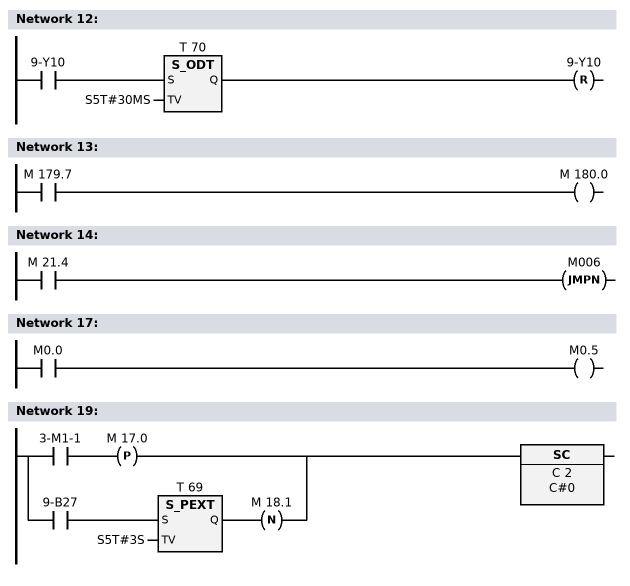
NETWORK
TITLE =
      A     "9-Y10";
      L     S5T#30MS;
      SD    T 70;
      NOP   0;
      NOP   0;
      NOP   0;
      A     T 70;
      R     "9-Y10";
NETWORK
TITLE =
      A     M 179.7;
      =     M 180.0;
NETWORK
TITLE =
      A     M 21.4;
      JCN   M006;
NETWORK
TITLE =
      L     MD 176;
      CAD;
      SLD   1;
      CAD;
      T     MD 176;
NETWORK
TITLE =
      L     MD 180;
      CAD;
      SLD   1;
      CAD;
      T     MD 180;
NETWORK
TITLE =
M006: A     "М0.0";
      =     "М0.5";
NETWORK
TITLE =
      A(;
      A     M 245.6;
      S     M 18.4;
      A(;
      O     "5-S11";
      O     M 245.3;
      ON    "М100.4";
      );
      R     M 18.4;
      A     M 18.4;
      );
      FN    M 18.2;
      R     M 18.0;
NETWORK
TITLE =
      A     "3-М1-1";
      FP    M 17.0;
      O(;
      A(;
      A     "9-В27";
      L     S5T#3S;
      SE    T 69;
      NOP   0;
      NOP   0;
      NOP   0;
      A     T 69;
      );
      FN    M 18.1;
      );
      L     C#0;
      S     C 2;
END_FUNCTION

FUNCTION FC 66 : VOID
AUTHOR : Stolz
VERSION : 0.1
BEGIN
// (block stored without names or comments; labels and parameter names are numbered)
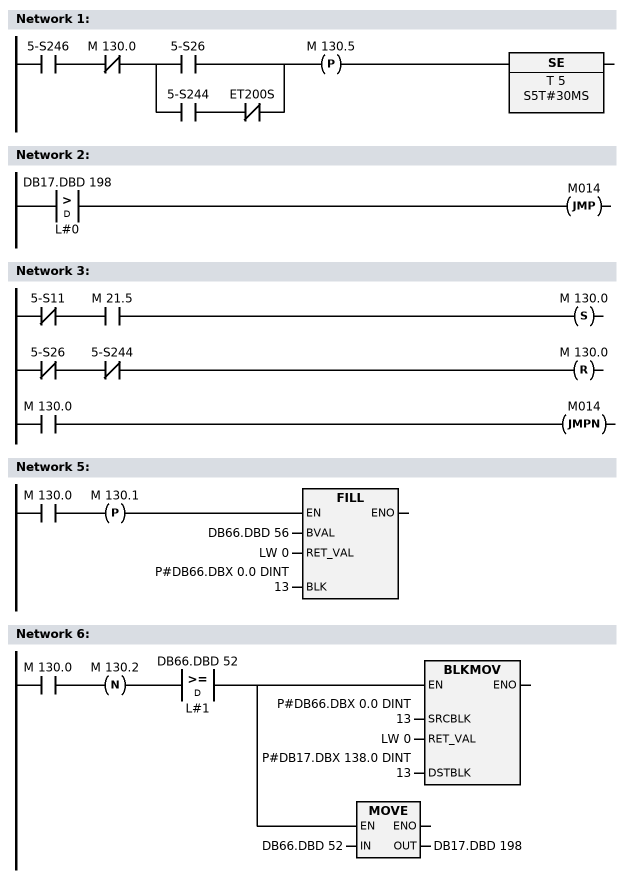
NETWORK
TITLE =
      A     "5-S246";
      AN    M 130.0;
      A(;
      O     "5-S26";
      O;
      A     "5-S244";
      AN    "ET200S";
      );
      FP    M 130.5;
      L     S5T#30MS;
      SE    T 5;
NETWORK
TITLE =
      L     DB17.DBD 198;
      L     L#0;
      >D;
      JC    M014;
NETWORK
TITLE =
      AN    "5-S11";
      A     M 21.5;
      S     M 130.0;
      AN    "5-S26";
      AN    "5-S244";
      R     M 130.0;
      A     M 130.0;
      JCN   M014;
NETWORK
TITLE =
      A     M 21.7;
      JCN   M001;
      L     C 10;
      ITD;
      T     DB66.DBD 0;
      L     L#0;
      T     DB66.DBD 52;
M001: A     M 22.0;
      JCN   M002;
      L     C 10;
      ITD;
      T     DB66.DBD 4;
      L     L#0;
      T     DB66.DBD 52;
M002: A     M 22.1;
      JCN   M003;
      L     C 10;
      ITD;
      T     DB66.DBD 8;
      L     L#0;
      T     DB66.DBD 52;
M003: A     M 22.2;
      JCN   M004;
      L     C 10;
      ITD;
      T     DB66.DBD 12;
      L     L#0;
      T     DB66.DBD 52;
M004: A     M 22.3;
      JCN   M005;
      L     C 10;
      ITD;
      T     DB66.DBD 16;
      L     L#0;
      T     DB66.DBD 52;
M005: A     M 22.4;
      JCN   M006;
      L     C 10;
      ITD;
      T     DB66.DBD 20;
      L     L#0;
      T     DB66.DBD 52;
M006: A     M 22.5;
      JCN   M007;
      L     C 10;
      ITD;
      T     DB66.DBD 24;
      L     L#0;
      T     DB66.DBD 52;
M007: A     M 24.0;
      JCN   M008;
      L     C 10;
      ITD;
      T     DB66.DBD 28;
      L     L#0;
      T     DB66.DBD 52;
M008: A     M 24.1;
      JCN   M009;
      L     C 10;
      ITD;
      T     DB66.DBD 32;
      L     L#0;
      T     DB66.DBD 52;
M009: A     M 24.2;
      JCN   M010;
      L     C 10;
      ITD;
      T     DB66.DBD 36;
      L     L#0;
      T     DB66.DBD 52;
M010: A     M 24.3;
      JCN   M011;
      L     C 10;
      ITD;
      T     DB66.DBD 40;
      L     L#0;
      T     DB66.DBD 52;
M011: A     M 24.4;
      JCN   M012;
      L     C 10;
      ITD;
      T     DB66.DBD 44;
      L     L#0;
      T     DB66.DBD 52;
M012: A     M 24.5;
      JCN   M013;
      L     C 10;
      ITD;
      T     DB66.DBD 48;
      L     L#0;
      T     DB66.DBD 52;
M013: A     M 21.6;
      JCN   M014;
      L     C 10;
      ITD;
      T     DB66.DBD 52;
NETWORK
TITLE =
M014: A     M 130.0;
      FP    M 130.1;
      JNB   M015;
      CALL  "FILL" (
           BVAL                     := DB66.DBD 56,
           RET_VAL                  := LW 0,
           BLK                      := P#DB66.DBX 0.0 DINT 13);
M015: NOP   0;
NETWORK
TITLE =
      A     M 130.0;
      FN    M 130.2;
      A(;
      L     DB66.DBD 52;
      L     L#1;
      >=D;
      );
      =     L 2.0;
      A     L 2.0;
      JNB   M016;
      CALL  "BLKMOV" (
           SRCBLK                   := P#DB66.DBX 0.0 DINT 13,
           RET_VAL                  := LW 0,
           DSTBLK                   := P#DB17.DBX 138.0 DINT 13);
M016: NOP   0;
      A     L 2.0;
      JNB   M017;
      L     DB66.DBD 52;
      T     DB17.DBD 198;
M017: NOP   0;
END_FUNCTION

FUNCTION FC 100 : VOID
AUTHOR : Stolz
VERSION : 0.1
BEGIN
// (block stored without names or comments; labels and parameter names are numbered)
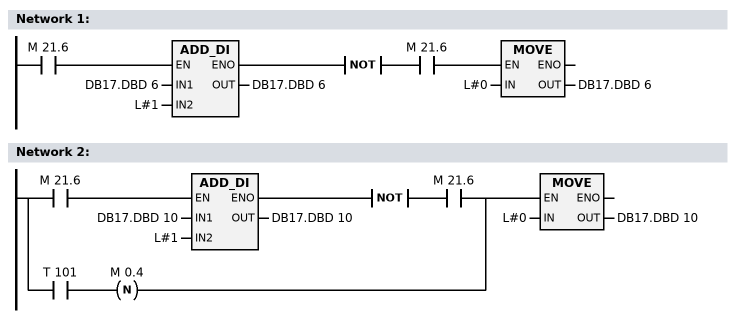
NETWORK
TITLE =
      A(;
      A     M 21.6;
      JNB   M001;
      L     DB17.DBD 6;
      L     L#1;
      +D;
      T     DB17.DBD 6;
      AN    OV;
      SAVE;
      CLR;
M001: A     BR;
      );
      NOT;
      A     M 21.6;
      JNB   M002;
      L     L#0;
      T     DB17.DBD 6;
M002: NOP   0;
NETWORK
TITLE =
      A(;
      A(;
      A     M 21.6;
      JNB   M003;
      L     DB17.DBD 10;
      L     L#1;
      +D;
      T     DB17.DBD 10;
      AN    OV;
      SAVE;
      CLR;
M003: A     BR;
      );
      NOT;
      A     M 21.6;
      O(;
      A     T 101;
      FN    M 0.4;
      );
      );
      JNB   M004;
      L     L#0;
      T     DB17.DBD 10;
M004: NOP   0;
END_FUNCTION

FUNCTION FC 104 : VOID
AUTHOR : Stolz
NAME : IstUmin
VERSION : 0.1
BEGIN
// (block stored without names or comments; labels and parameter names are numbered)
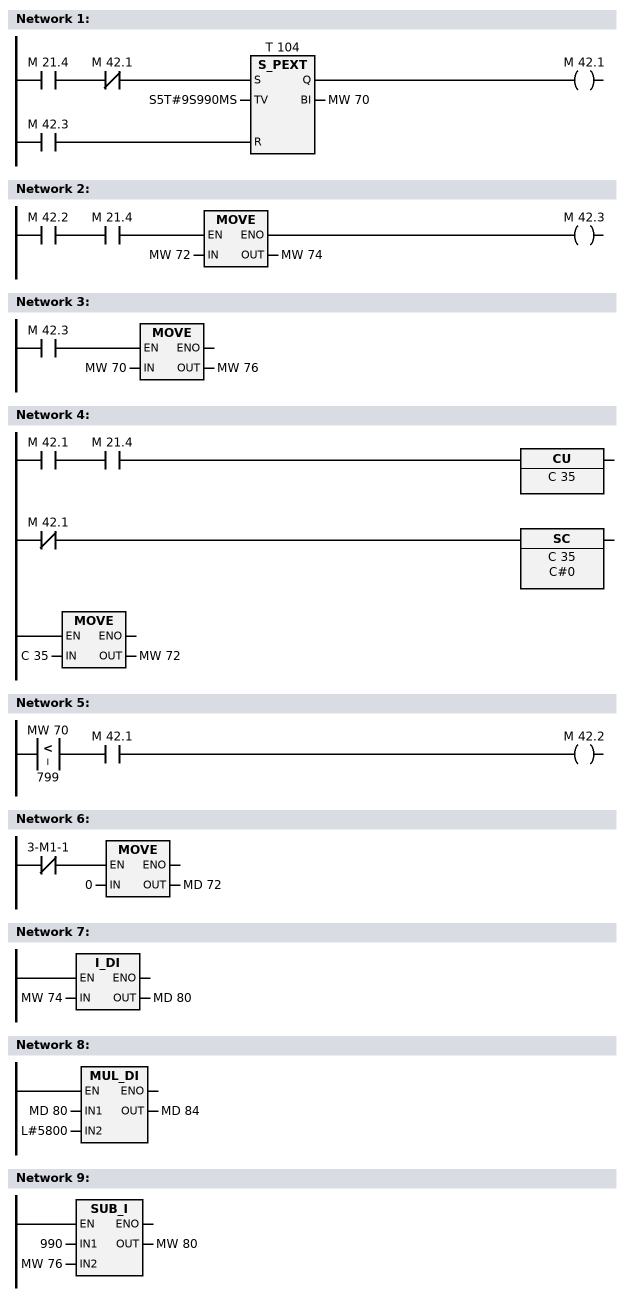
NETWORK
TITLE =
      A     M 21.4;
      AN    M 42.1;
      L     S5T#9S990MS;
      SE    T 104;
      A     M 42.3;
      R     T 104;
      L     T 104;
      T     MW 70;
      NOP   0;
      A     T 104;
      =     M 42.1;
NETWORK
TITLE =
      A     M 42.2;
      A     M 21.4;
      JNB   M001;
      L     MW 72;
      T     MW 74;
      SET;
      SAVE;
      CLR;
M001: A     BR;
      =     M 42.3;
NETWORK
TITLE =
      A     M 42.3;
      JNB   M002;
      L     MW 70;
      T     MW 76;
M002: NOP   0;
NETWORK
TITLE =
      A     M 42.1;
      A     M 21.4;
      CU    C 35;
      BLD   101;
      AN    M 42.1;
      L     C#0;
      S     C 35;
      NOP   0;
      L     C 35;
      T     MW 72;
      NOP   0;
      NOP   0;
NETWORK
TITLE =
      A(;
      L     MW 70;
      L     799;
      <I;
      );
      A     M 42.1;
      =     M 42.2;
NETWORK
TITLE =
      AN    "3-М1-1";
      JNB   M003;
      L     0;
      T     MD 72;
M003: NOP   0;
NETWORK
TITLE =
      L     MW 74;
      ITD;
      T     MD 80;
      NOP   0;
NETWORK
TITLE =
      L     MD 80;
      L     L#5800;
      *D;
      T     MD 84;
      NOP   0;
NETWORK
TITLE =
      L     990;
      L     MW 76;
      -I;
      T     MW 80;
      NOP   0;
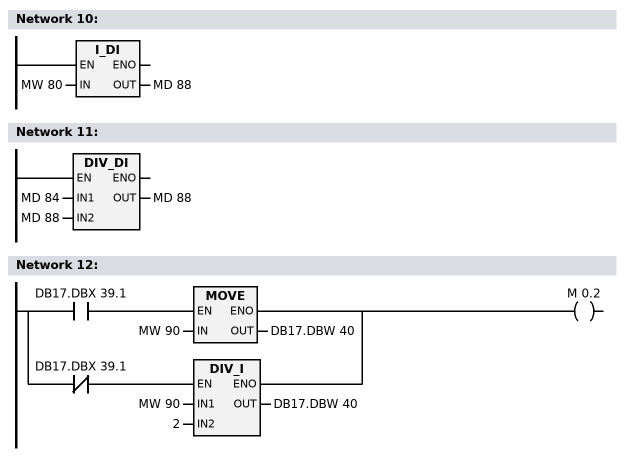
NETWORK
TITLE =
      L     MW 80;
      ITD;
      T     MD 88;
      NOP   0;
NETWORK
TITLE =
      L     MD 84;
      L     MD 88;
      /D;
      T     MD 88;
      NOP   0;
NETWORK
TITLE =
      O(;
      A     DB17.DBX 39.1;
      JNB   M004;
      L     MW 90;
      T     DB17.DBW 40;
      SET;
      SAVE;
      CLR;
M004: A     BR;
      );
      O(;
      AN    DB17.DBX 39.1;
      JNB   M005;
      L     MW 90;
      L     2;
      /I;
      T     DB17.DBW 40;
      AN    OV;
      SAVE;
      CLR;
M005: A     BR;
      );
      =     M 0.2;
END_FUNCTION

FUNCTION FC 105 : VOID
AUTHOR : Stolz
NAME : SollUmin
VERSION : 0.2
VAR_TEMP
  TEMP0 : INT ;
  TEMP1 : DINT ;
  TEMP2 : DINT ;
  TEMP3 : DINT ;
  TEMP4 : INT ;
  TEMP5 : DINT ;
  TEMP6 : DINT ;
  TEMP7 : DINT ;
END_VAR
BEGIN
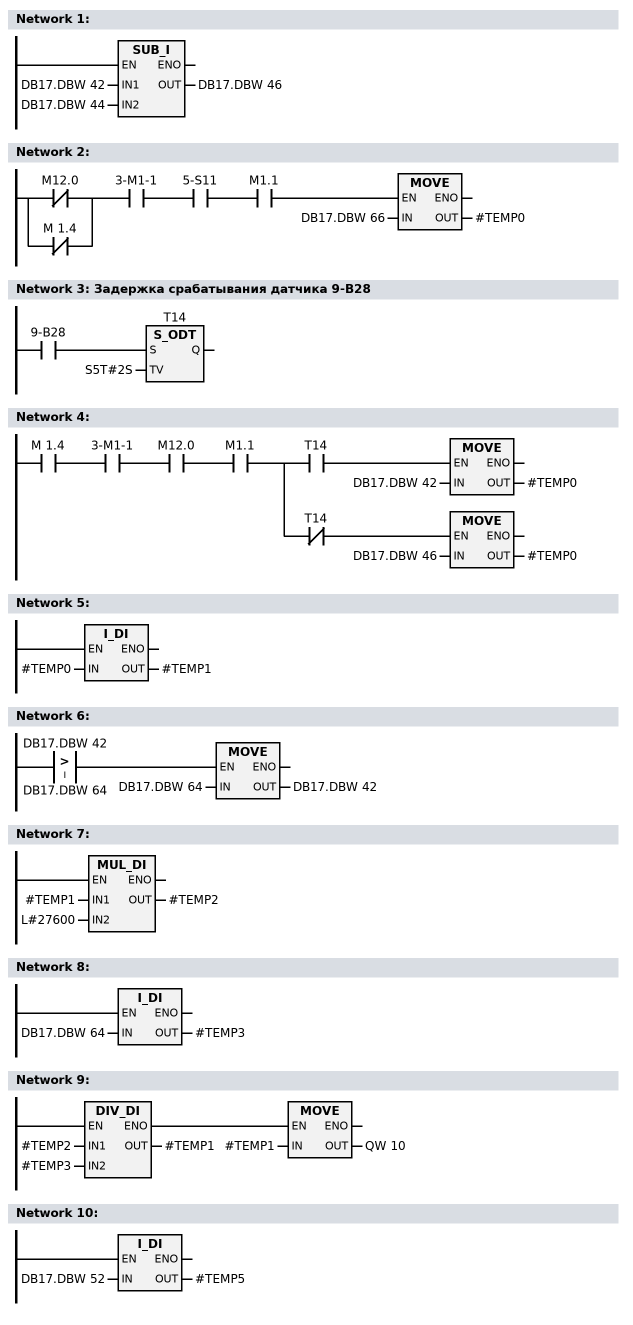
NETWORK
TITLE =
      L     DB17.DBW 42;
      L     DB17.DBW 44;
      -I;
      T     DB17.DBW 46;
      NOP   0;
NETWORK
TITLE =
      A(;
      ON    "М12.0";
      ON    M 1.4;
      );
      A     "3-М1-1";
      A     "5-S11";
      A     "М1.1";
      JNB   _001;
      L     DB17.DBW 66;
      T     #TEMP0;
_001: NOP   0;
NETWORK
TITLE = Задержка срабатывания датчика 9-В28
      A     "9-В28";
      L     S5T#2S;
      SD    "Т14";
      NOP   0;
      NOP   0;
      NOP   0;
      NOP   0;
NETWORK
TITLE =
      A     M 1.4;
      A     "3-М1-1";
      A     "М12.0";
      A     "М1.1";
      =     L 28.0;
      A     L 28.0;
      A     "Т14";
      JNB   _002;
      L     DB17.DBW 42;
      T     #TEMP0;
_002: NOP   0;
      A     L 28.0;
      AN    "Т14";
      JNB   _003;
      L     DB17.DBW 46;
      T     #TEMP0;
_003: NOP   0;
NETWORK
TITLE =
      L     #TEMP0;
      ITD;
      T     #TEMP1;
      NOP   0;
NETWORK
TITLE =
      A(;
      L     DB17.DBW 42;
      L     DB17.DBW 64;
      >I;
      );
      JNB   _004;
      L     DB17.DBW 64;
      T     DB17.DBW 42;
_004: NOP   0;
NETWORK
TITLE =
      L     #TEMP1;
      L     L#27600;
      *D;
      T     #TEMP2;
      NOP   0;
NETWORK
TITLE =
      L     DB17.DBW 64;
      ITD;
      T     #TEMP3;
      NOP   0;
NETWORK
TITLE =
      A(;
      L     #TEMP2;
      L     #TEMP3;
      /D;
      T     #TEMP1;
      AN    OV;
      SAVE;
      CLR;
      A     BR;
      );
      JNB   _005;
      L     #TEMP1;
      T     QW 10;
_005: NOP   0;
NETWORK
TITLE =
      L     DB17.DBW 52;
      ITD;
      T     #TEMP5;
      NOP   0;
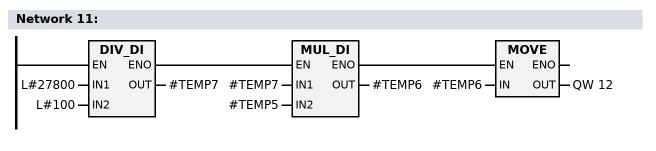
NETWORK
TITLE =
      A(;
      A(;
      L     L#27800;
      L     L#100;
      /D;
      T     #TEMP7;
      AN    OV;
      SAVE;
      CLR;
      A     BR;
      );
      JNB   _006;
      L     #TEMP7;
      L     #TEMP5;
      *D;
      T     #TEMP6;
      AN    OV;
      SAVE;
      CLR;
_006: A     BR;
      );
      JNB   _007;
      L     #TEMP6;
      T     QW 12;
_007: NOP   0;
END_FUNCTION

FUNCTION FC 110 : VOID
AUTHOR : Joehring
VERSION : 0.1
BEGIN
// (block stored without names or comments; labels and parameter names are numbered)
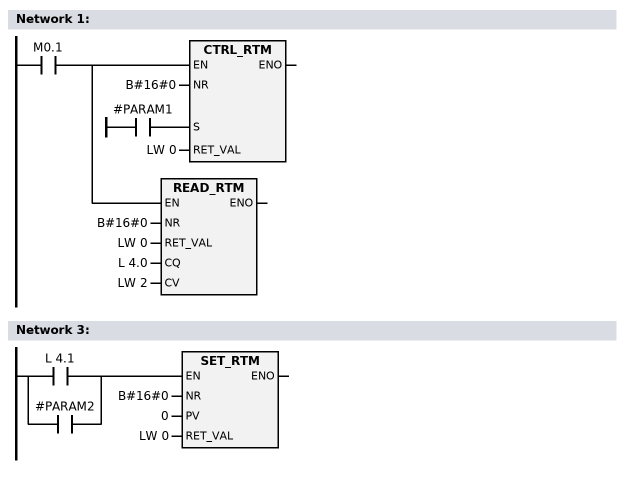
NETWORK
TITLE =
      A     "М0.1";
      =     L 5.0;
      A     #PARAM1;
      =     L 5.1;
      BLD   103;
      A     L 5.0;
      JNB   M001;
      CALL  "CTRL_RTM" (
           NR                       := B#16#0,
           S                        := L 5.1,
           RET_VAL                  := LW 0);
M001: NOP   0;
      A     L 5.0;
      JNB   M002;
      CALL  "READ_RTM" (
           NR                       := B#16#0,
           RET_VAL                  := LW 0,
           CQ                       := L 4.0,
           CV                       := LW 2);
M002: NOP   0;
NETWORK
TITLE =
      L     LW 2;
      L     1;
      >=I;
      =     L 4.1;
NETWORK
TITLE =
      A(;
      O     L 4.1;
      O     #PARAM2;
      );
      JNB   M003;
      CALL  "SET_RTM" (
           NR                       := B#16#0,
           PV                       := 0,
           RET_VAL                  := LW 0);
M003: NOP   0;
NETWORK
TITLE =
      O(;
      A     L 4.1;
      JNB   M004;
      L     #PARAM3;
      L     L#1;
      +D;
      T     #PARAM3;
      AN    OV;
      SAVE;
      CLR;
M004: A     BR;
      );
      O(;
      A     #PARAM2;
      JNB   M005;
      L     0;
      T     #PARAM3;
      SET;
      SAVE;
      CLR;
M005: A     BR;
      );
      =     L 4.2;
END_FUNCTION

// FC 125: know-how protected block, not included

DATA_BLOCK DB 17
AUTHOR : Stolz
VERSION : 0.2
BEGIN
// 360 bytes; values not shown
END_DATA_BLOCK

DATA_BLOCK DB 66
AUTHOR : Stolz
VERSION : 0.0
BEGIN
// 60 bytes; values not shown
END_DATA_BLOCK

DATA_BLOCK DB 77
AUTHOR : Stolz
VERSION : 0.0
BEGIN
// 80 bytes; values not shown
END_DATA_BLOCK

DATA_BLOCK DB 100
AUTHOR : Joehring
VERSION : 0.1
FB 100
BEGIN
END_DATA_BLOCK

DATA_BLOCK DB 111
VERSION : 0.1
BEGIN
// 88 bytes; values not shown
END_DATA_BLOCK

DATA_BLOCK DB 125
VERSION : 0.0
FB 125
BEGIN
END_DATA_BLOCK

ORGANIZATION_BLOCK OB 1
AUTHOR : Stolz
VERSION : 0.1
BEGIN
// (block stored without names or comments; labels and parameter names are numbered)
NETWORK
TITLE =
      UC    FC 50;
NETWORK
TITLE =
      UC    "FC2";
NETWORK
TITLE =
      UC    "FC3";
NETWORK
TITLE =
      UC    "FC4";
NETWORK
TITLE =
      UC    "FC6";
NETWORK
TITLE =
      UC    "FC7";
NETWORK
TITLE =
      UC    FC 10;
NETWORK
TITLE =
      UC    FC 11;
NETWORK
TITLE =
      UC    FC 12;
NETWORK
TITLE =
      UC    FC 23;
NETWORK
TITLE =
      UC    FC 24;
NETWORK
TITLE =
      UC    FC 60;
NETWORK
TITLE =
      A     DB17.DBX 39.3;
      CC    FC 61;
NETWORK
TITLE =
      UC    FC 100;
NETWORK
TITLE =
      UC    FC 104;
NETWORK
TITLE =
      UC    FC 105;
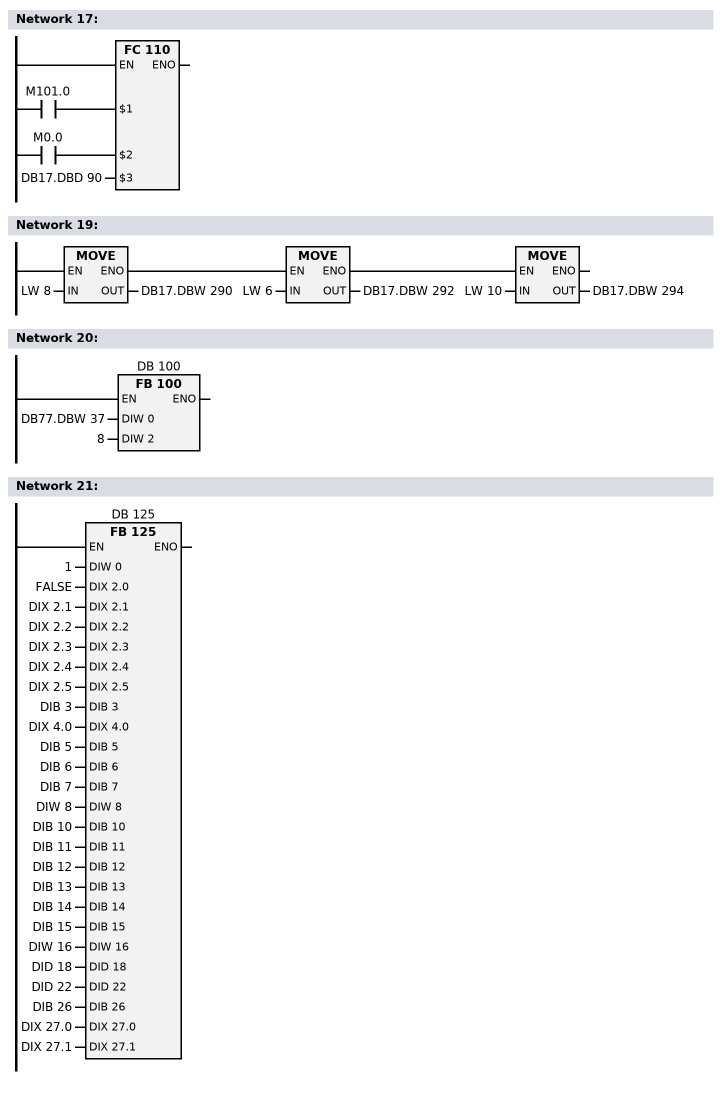
NETWORK
TITLE =
      A     "М101.0";
      =     L 20.0;
      BLD   103;
      A     "М0.0";
      =     L 20.1;
      BLD   103;
      CALL  FC 110 (
           $1                       := L 20.0,
           $2                       := L 20.1,
           $3                       := DB17.DBD 90);
      NOP   0;
NETWORK
TITLE =
      UC    FC 66;
NETWORK
TITLE =
      A(;
      A(;
      L     LW 8;
      T     DB17.DBW 290;
      SET;
      SAVE;
      CLR;
      A     BR;
      );
      JNB   M001;
      L     LW 6;
      T     DB17.DBW 292;
      SET;
      SAVE;
      CLR;
M001: A     BR;
      );
      JNB   M002;
      L     LW 10;
      T     DB17.DBW 294;
M002: NOP   0;
NETWORK
TITLE =
      CALL  FB 100 , DB 100 (
           DIW 0                    := DB77.DBW 37,
           DIW 2                    := 8);
      NOP   0;
NETWORK
TITLE =
      CALL  FB 125 , DB 125 (
           DIW 0                    := 1,
           DIX 2.0                  := FALSE,
           DIX 2.1                  := DIX 2.1,
           DIX 2.2                  := DIX 2.2,
           DIX 2.3                  := DIX 2.3,
           DIX 2.4                  := DIX 2.4,
           DIX 2.5                  := DIX 2.5,
           DIB 3                    := DIB 3,
           DIX 4.0                  := DIX 4.0,
           DIB 5                    := DIB 5,
           DIB 6                    := DIB 6,
           DIB 7                    := DIB 7,
           DIW 8                    := DIW 8,
           DIB 10                   := DIB 10,
           DIB 11                   := DIB 11,
           DIB 12                   := DIB 12,
           DIB 13                   := DIB 13,
           DIB 14                   := DIB 14,
           DIB 15                   := DIB 15,
           DIW 16                   := DIW 16,
           DID 18                   := DID 18,
           DID 22                   := DID 22,
           DIB 26                   := DIB 26,
           DIX 27.0                 := DIX 27.0,
           DIX 27.1                 := DIX 27.1);
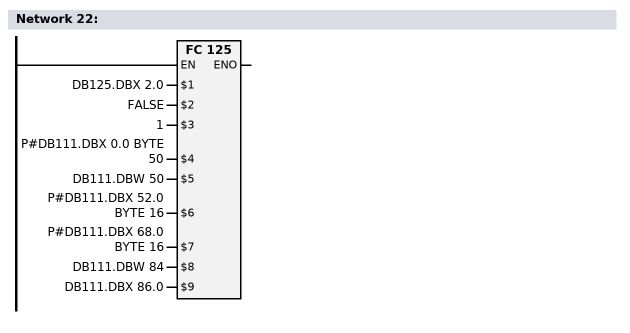
NETWORK
TITLE =
      CALL  FC 125 (
           $1                       := DB125.DBX 2.0,
           $2                       := FALSE,
           $3                       := 1,
           $4                       := P#DB111.DBX 0.0 BYTE 50,
           $5                       := DB111.DBW 50,
           $6                       := P#DB111.DBX 52.0 BYTE 16,
           $7                       := P#DB111.DBX 68.0 BYTE 16,
           $8                       := DB111.DBW 84,
           $9                       := DB111.DBX 86.0);
END_ORGANIZATION_BLOCK

ORGANIZATION_BLOCK OB 40
AUTHOR : Stolz
VERSION : 0.1
BEGIN
// (block stored without names or comments; labels and parameter names are numbered)
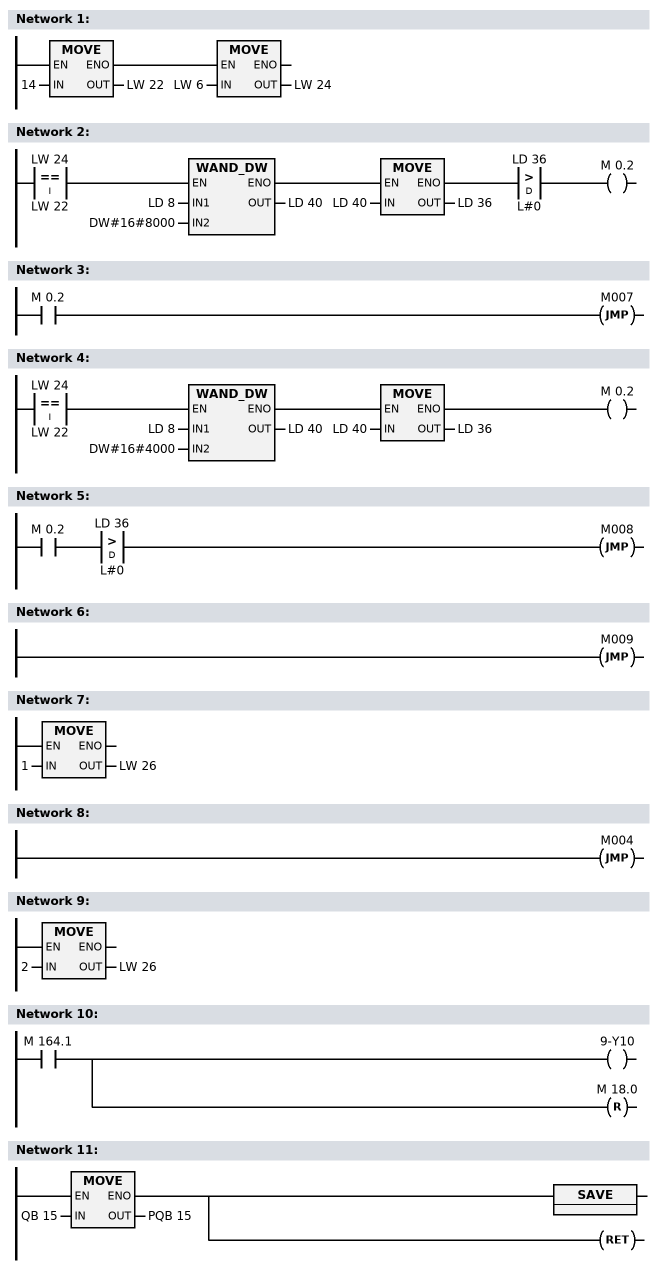
NETWORK
TITLE =
      A(;
      L     14;
      T     LW 22;
      SET;
      SAVE;
      CLR;
      A     BR;
      );
      JNB   M001;
      L     LW 6;
      T     LW 24;
M001: NOP   0;
NETWORK
TITLE =
      A(;
      A(;
      A(;
      L     LW 24;
      L     LW 22;
      ==I;
      );
      JNB   M002;
      L     LD 8;
      L     DW#16#8000;
      AD;
      T     LD 40;
      SET;
      SAVE;
      CLR;
M002: A     BR;
      );
      JNB   M003;
      L     LD 40;
      T     LD 36;
      SET;
      SAVE;
      CLR;
M003: A     BR;
      );
      A(;
      L     LD 36;
      L     L#0;
      >D;
      );
      =     M 0.2;
NETWORK
TITLE =
      A     M 0.2;
      JC    M007;
NETWORK
TITLE =
M004: A(;
      A(;
      L     LW 24;
      L     LW 22;
      ==I;
      );
      JNB   M005;
      L     LD 8;
      L     DW#16#4000;
      AD;
      T     LD 40;
      SET;
      SAVE;
      CLR;
M005: A     BR;
      );
      JNB   M006;
      L     LD 40;
      T     LD 36;
      SET;
      SAVE;
      CLR;
M006: A     BR;
      =     M 0.2;
NETWORK
TITLE =
      A     M 0.2;
      A(;
      L     LD 36;
      L     L#0;
      >D;
      );
      JC    M008;
NETWORK
TITLE =
      JU    M009;
NETWORK
TITLE =
M007: L     1;
      T     LW 26;
      NOP   0;
NETWORK
TITLE =
      JU    M004;
NETWORK
TITLE =
M008: L     2;
      T     LW 26;
      NOP   0;
NETWORK
TITLE =
      A     M 164.1;
      =     "9-Y10";
      R     M 18.0;
NETWORK
TITLE =
M009: L     QB 15;
      T     PQB 15;
      SET;
      SAVE;
      CLR;
      A     BR;
      SAVE;
      BEC;
END_ORGANIZATION_BLOCK

ORGANIZATION_BLOCK OB 80
AUTHOR : Ham
FAMILY : XOMAT
VERSION : 1.1
BEGIN
// (block stored without names or comments; labels and parameter names are numbered)
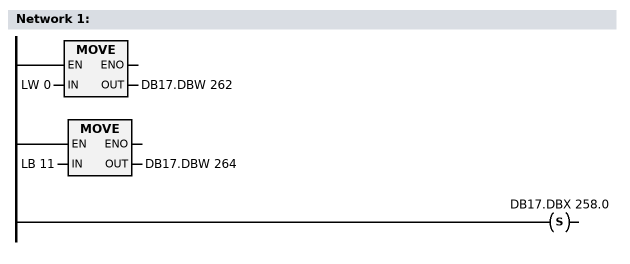
NETWORK
TITLE =
      L     LW 0;
      T     DB17.DBW 262;
      L     LB 11;
      T     DB17.DBW 264;
      SET;
      S     DB17.DBX 258.0;
END_ORGANIZATION_BLOCK

ORGANIZATION_BLOCK OB 82
AUTHOR : Ham
FAMILY : XOMAT
VERSION : 1.1
BEGIN
// (block stored without names or comments; labels and parameter names are numbered)
NETWORK
TITLE =
      L     LW 6;
      T     DB17.DBW 268;
      L     LW 0;
      T     DB17.DBW 266;
      L     W#16#3942;
      ==I;
      =     DB17.DBX 258.2;
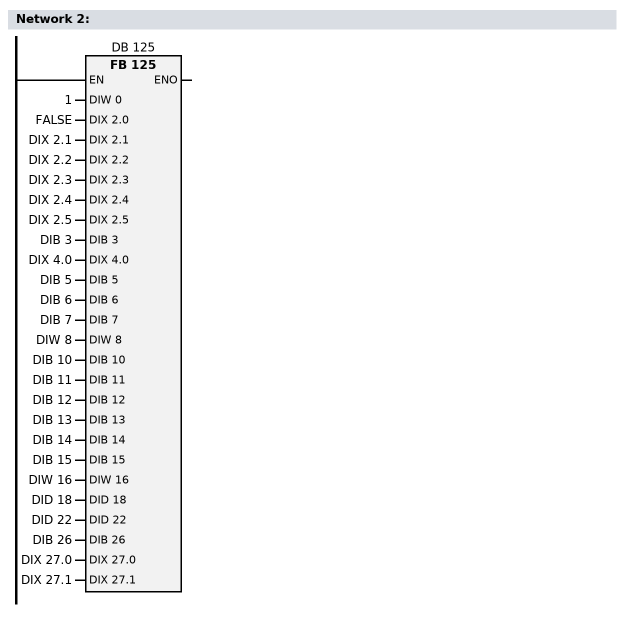
NETWORK
TITLE =
      CALL  FB 125 , DB 125 (
           DIW 0                    := 1,
           DIX 2.0                  := FALSE,
           DIX 2.1                  := DIX 2.1,
           DIX 2.2                  := DIX 2.2,
           DIX 2.3                  := DIX 2.3,
           DIX 2.4                  := DIX 2.4,
           DIX 2.5                  := DIX 2.5,
           DIB 3                    := DIB 3,
           DIX 4.0                  := DIX 4.0,
           DIB 5                    := DIB 5,
           DIB 6                    := DIB 6,
           DIB 7                    := DIB 7,
           DIW 8                    := DIW 8,
           DIB 10                   := DIB 10,
           DIB 11                   := DIB 11,
           DIB 12                   := DIB 12,
           DIB 13                   := DIB 13,
           DIB 14                   := DIB 14,
           DIB 15                   := DIB 15,
           DIW 16                   := DIW 16,
           DID 18                   := DID 18,
           DID 22                   := DID 22,
           DIB 26                   := DIB 26,
           DIX 27.0                 := DIX 27.0,
           DIX 27.1                 := DIX 27.1);
END_ORGANIZATION_BLOCK

ORGANIZATION_BLOCK OB 85
AUTHOR : Ham
FAMILY : XOMAT
VERSION : 1.1
BEGIN
// (block stored without names or comments; labels and parameter names are numbered)
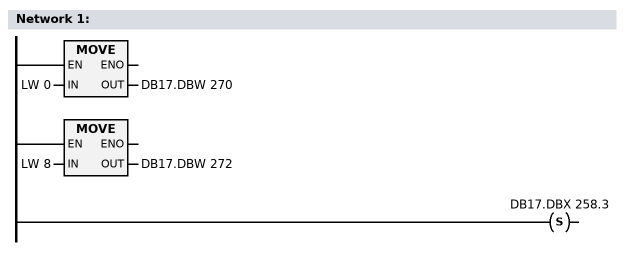
NETWORK
TITLE =
      L     LW 0;
      T     DB17.DBW 270;
      L     LW 8;
      T     DB17.DBW 272;
      SET;
      S     DB17.DBX 258.3;
END_ORGANIZATION_BLOCK

ORGANIZATION_BLOCK OB 86
AUTHOR : Ham
FAMILY : XOMAT
VERSION : 1.1
BEGIN
// (block stored without names or comments; labels and parameter names are numbered)
NETWORK
TITLE =
      L     0;
      T     DB17.DBW 276;
      L     LW 0;
      T     DB17.DBW 274;
      AW    W#16#FF;
      L     B#16#C4;
      ==I;
      JCN   M001;
      L     LB 11;
      T     DB17.DBW 276;
M001: L     LB 0;
      L     B#16#39;
      ==I;
      =     DB17.DBX 258.4;
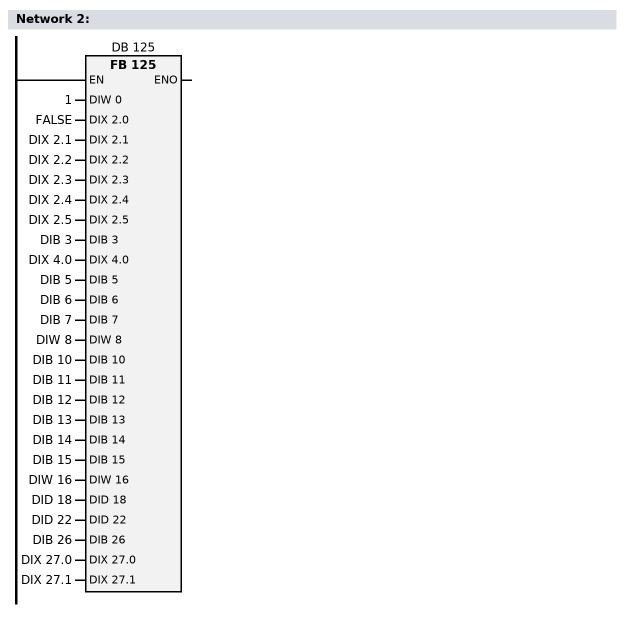
NETWORK
TITLE =
      CALL  FB 125 , DB 125 (
           DIW 0                    := 1,
           DIX 2.0                  := FALSE,
           DIX 2.1                  := DIX 2.1,
           DIX 2.2                  := DIX 2.2,
           DIX 2.3                  := DIX 2.3,
           DIX 2.4                  := DIX 2.4,
           DIX 2.5                  := DIX 2.5,
           DIB 3                    := DIB 3,
           DIX 4.0                  := DIX 4.0,
           DIB 5                    := DIB 5,
           DIB 6                    := DIB 6,
           DIB 7                    := DIB 7,
           DIW 8                    := DIW 8,
           DIB 10                   := DIB 10,
           DIB 11                   := DIB 11,
           DIB 12                   := DIB 12,
           DIB 13                   := DIB 13,
           DIB 14                   := DIB 14,
           DIB 15                   := DIB 15,
           DIW 16                   := DIW 16,
           DID 18                   := DID 18,
           DID 22                   := DID 22,
           DIB 26                   := DIB 26,
           DIX 27.0                 := DIX 27.0,
           DIX 27.1                 := DIX 27.1);
END_ORGANIZATION_BLOCK

ORGANIZATION_BLOCK OB 100
//Теплый пуск-сброс системной памяти.
AUTHOR : Stolz
NAME : Anlauf
VERSION : 0.1
VAR_TEMP
  TEMP0 : BYTE ;
  TEMP1 : BYTE ;
  TEMP2 : BYTE ;
  TEMP3 : BYTE ;
  TEMP4 : BYTE ;
  TEMP5 : BYTE ;
  TEMP6 : WORD ;
  TEMP7 : DWORD ;
  TEMP8 : DATE_AND_TIME ;
END_VAR
BEGIN
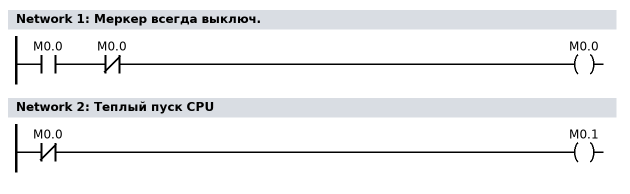
NETWORK
TITLE = Меркер всегда выключ.
      A     "М0.0";
      AN    "М0.0";
      =     "М0.0";
NETWORK
TITLE = Теплый пуск CPU
      AN    "М0.0";
      =     "М0.1";
END_ORGANIZATION_BLOCK

ORGANIZATION_BLOCK OB 121
//Блок обработки синхронных ошибок в прикладной программе
AUTHOR : Ham
FAMILY : XOMAT
VERSION : 1.1
VAR_TEMP
  TEMP0 : BYTE ;
  TEMP1 : BYTE ;
  TEMP2 : BYTE ;
  TEMP3 : BYTE ;
  TEMP4 : BYTE ;
  TEMP5 : BYTE ;
  TEMP6 : WORD ;
  TEMP7 : WORD ;
  TEMP8 : WORD ;
  TEMP9 : DATE_AND_TIME ;
END_VAR
BEGIN
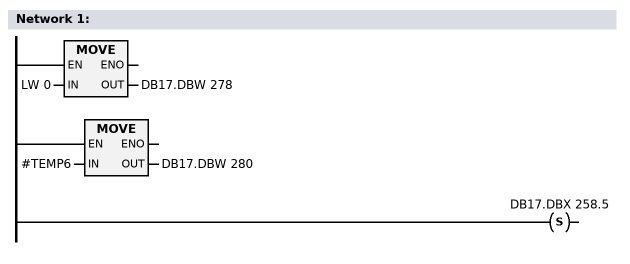
NETWORK
TITLE =
      L     LW 0;
      T     DB17.DBW 278;
      L     #TEMP6;
      T     DB17.DBW 280;
      SET;
      S     DB17.DBX 258.5;
END_ORGANIZATION_BLOCK

ORGANIZATION_BLOCK OB 122
//Блок обработки синхронных ошибок доступа к переферии.
AUTHOR : Ham
FAMILY : XOMAT
VERSION : 1.1
VAR_TEMP
  TEMP0 : BYTE ;
  TEMP1 : BYTE ;
  TEMP2 : BYTE ;
  TEMP3 : BYTE ;
  TEMP4 : BYTE ;
  TEMP5 : BYTE ;
  TEMP6 : WORD ;
  TEMP7 : WORD ;
  TEMP8 : WORD ;
  TEMP9 : DATE_AND_TIME ;
END_VAR
BEGIN
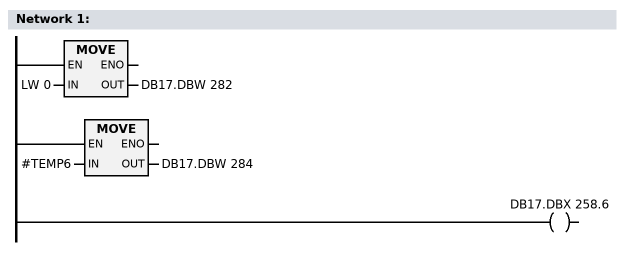
NETWORK
TITLE =
      L     LW 0;
      T     DB17.DBW 282;
      L     #TEMP6;
      T     DB17.DBW 284;
      SET;
      =     DB17.DBX 258.6;
END_ORGANIZATION_BLOCK
